// TIA Portal V16 export
// export: Created 2022-11-17T11:55:13.2880017Z, ExportSetting WithDefaults, DisplayName Totally Integrated Automation Portal, DisplayVersion V16 Update 6, DisplayName TIA Portal Version Control Interface, DisplayVersion V16 Update 2, DisplayName TIA Portal Openness, DisplayVersion V16 Update 6, DisplayName SINAMICS Startdrive Advanced, DisplayVersion V16 Update 5, DisplayName SINAMICS Startdrive G130, G150, S120, S150, SINAMICS MV, S210, DisplayVersion V16 Update 5, DisplayName SINAMICS Startdrive G110M, G120, G120C, G120D, G120P, G115D, DisplayVersion V16 Update 5, DisplayName STEP 7 Professional, DisplayVersion V16 Update 6, DisplayName STEP 7 Safety, DisplayVersion V16, DisplayName WinCC Advanced, DisplayVersion V16 Update 6
FUNCTION "FC37_MultiprogramSignal" : Void   // FC37, LAD
TITLE = Multiprogram with program selection by external signal
{ S7_Optimized_Access := 'FALSE' }
AUTHOR : Robopac
VERSION : 0.0
// stored: AutoNumber false, IsIECCheckEnabled false, SetENOAutomatically false, UDAEnableTagReadback false
   VAR_TEMP   // added for the SCL form of the ladder/FBD networks
      _w1 : Bool;
   END_VAR
BEGIN

REGION Network 1
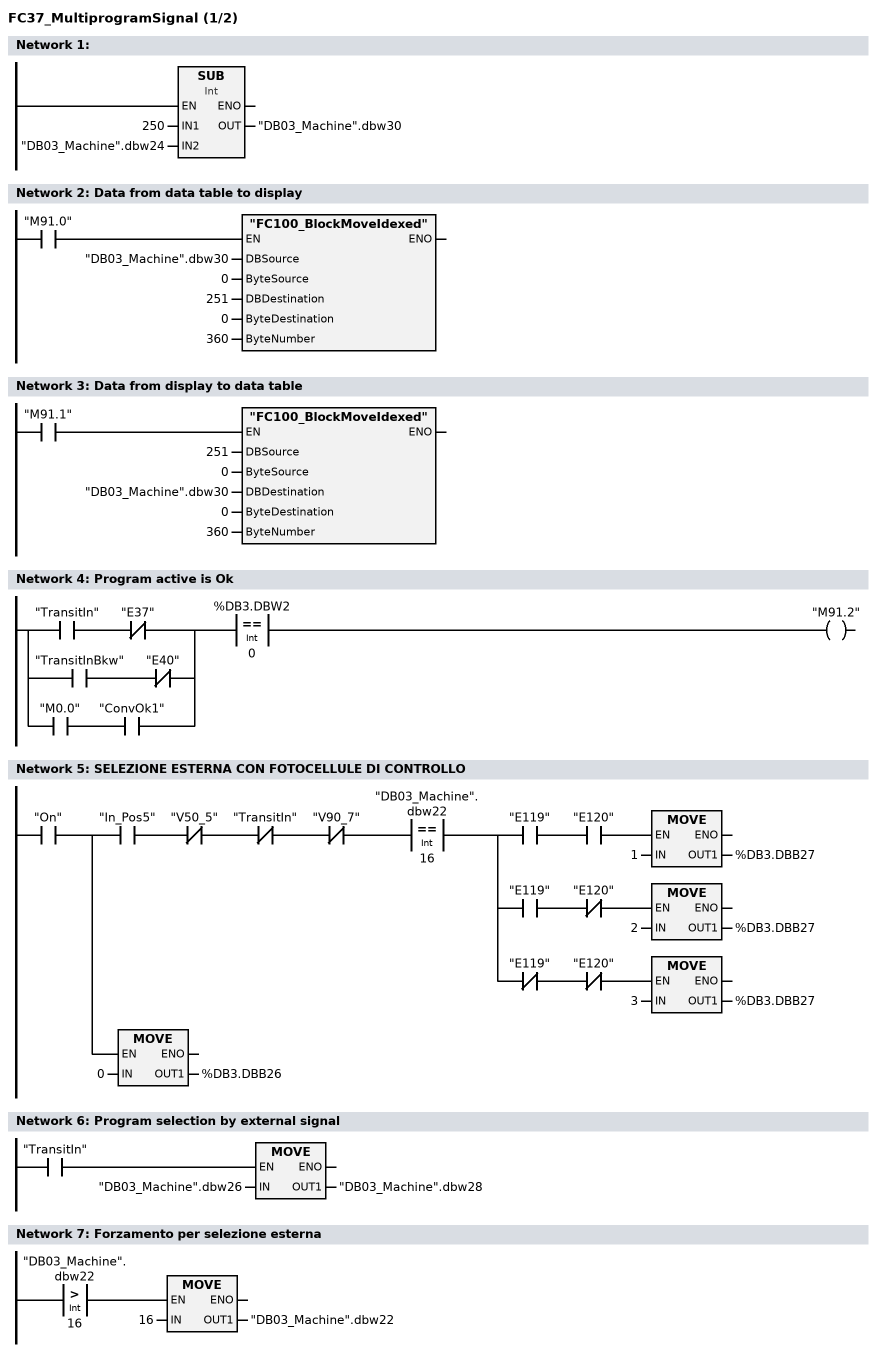
   RUNG wire#powerrail
      { S7_Templates := "SrcType := Int"; S7_GenerateENO := "TRUE" } Sub(in1 := 250, in2 := "DB03_Machine".dbw24, out => "DB03_Machine".dbw30)
   END_RUNG
   // the same network as SCL:
   "DB03_Machine".dbw30 := 250 - "DB03_Machine".dbw24;
END_REGION

REGION Network 2: Data from data table to display
   RUNG wire#powerrail
      Contact( "M91.0" )
      "FC100_BlockMoveIdexed"(DBSource := "DB03_Machine".dbw30, ByteSource := 0, DBDestination := 251, ByteDestination := 0, ByteNumber := 360)
   END_RUNG
   // the same network as SCL:
   IF "M91.0" THEN
       "FC100_BlockMoveIdexed"(DBSource := "DB03_Machine".dbw30,
                               ByteSource := 0,
                               DBDestination := 251,
                               ByteDestination := 0,
                               ByteNumber := 360);
   END_IF;
END_REGION

REGION Network 3: Data from display to data table
   RUNG wire#powerrail
      Contact( "M91.1" )
      "FC100_BlockMoveIdexed"(DBSource := 251, ByteSource := 0, DBDestination := "DB03_Machine".dbw30, ByteDestination := 0, ByteNumber := 360)
   END_RUNG
   // the same network as SCL:
   IF "M91.1" THEN
       "FC100_BlockMoveIdexed"(DBSource := 251,
                               ByteSource := 0,
                               DBDestination := "DB03_Machine".dbw30,
                               ByteDestination := 0,
                               ByteNumber := 360);
   END_IF;
END_REGION

REGION Network 4: Program active is Ok
   RUNG wire#powerrail
      Contact( "TransitIn" )
      I_Contact( "E37" )
      wire#w1
      { S7_Templates := "SrcType := Int" } EQ_Contact(in1 := %DB3.DBW2, in2 := 0)
      Coil( "M91.2" )
   END_RUNG
   RUNG wire#powerrail
      Contact( "TransitInBkw" )
      I_Contact( "E40" )
   END_RUNG wire#w1
   RUNG wire#powerrail
      Contact( "M0.0" )
      Contact( "ConvOk1" )
   END_RUNG wire#w1
   // the same network as SCL:
   "M91.2" := (("TransitIn" AND NOT "E37") OR ("TransitInBkw" AND NOT "E40") OR ("M0.0" AND "ConvOk1")) AND (%DB3.DBW2 = 0);
END_REGION

REGION Network 5: SELEZIONE ESTERNA CON FOTOCELLULE DI CONTROLLO
   RUNG wire#powerrail
      Contact( "On" )
      wire#w1
      Contact( "In_Pos5" )
      I_Contact( "V50_5" )
      I_Contact( "TransitIn" )
      I_Contact( "V90_7" )
      { S7_Templates := "SrcType := Int" } EQ_Contact(in1 := "DB03_Machine".dbw22, in2 := 16)
      wire#w2
      Contact( "E119" )
      Contact( "E120" )
      Move(in := 1, out1 => %DB3.DBB27)
   END_RUNG
   RUNG wire#w2
      Contact( "E119" )
      I_Contact( "E120" )
      Move(in := 2, out1 => %DB3.DBB27)
   END_RUNG
   RUNG wire#w2
      I_Contact( "E119" )
      I_Contact( "E120" )
      Move(in := 3, out1 => %DB3.DBB27)
   END_RUNG
   RUNG wire#w1
      { S7_GenerateENO := "TRUE" } Move(in := 0, out1 => %DB3.DBB26)
   END_RUNG
   // the same network as SCL:
   #_w1 := "On" AND "In_Pos5" AND NOT "V50_5" AND NOT "TransitIn" AND NOT "V90_7" AND ("DB03_Machine".dbw22 = 16);
   IF #_w1 AND "E119" AND "E120" THEN %DB3.DBB27 := 1; END_IF;
   IF #_w1 AND "E119" AND NOT "E120" THEN %DB3.DBB27 := 2; END_IF;
   IF #_w1 AND NOT "E119" AND NOT "E120" THEN %DB3.DBB27 := 3; END_IF;
   IF "On" THEN %DB3.DBB26 := 0; END_IF;
END_REGION

REGION Network 6: Program selection by external signal
   RUNG wire#powerrail
      Contact( "TransitIn" )
      { S7_GenerateENO := "TRUE" } Move(in := "DB03_Machine".dbw26, out1 => "DB03_Machine".dbw28)
   END_RUNG
   // the same network as SCL:
   IF "TransitIn" THEN "DB03_Machine".dbw28 := "DB03_Machine".dbw26; END_IF;
END_REGION

REGION Network 7: Forzamento per selezione esterna
   RUNG wire#powerrail
      { S7_Templates := "SrcType := Int" } GT_Contact(in1 := "DB03_Machine".dbw22, in2 := 16)
      { S7_GenerateENO := "TRUE" } Move(in := 16, out1 => "DB03_Machine".dbw22)
   END_RUNG
   // the same network as SCL:
   IF "DB03_Machine".dbw22 > 16 THEN "DB03_Machine".dbw22 := 16; END_IF;
END_REGION

REGION Network 8: Program selection by display
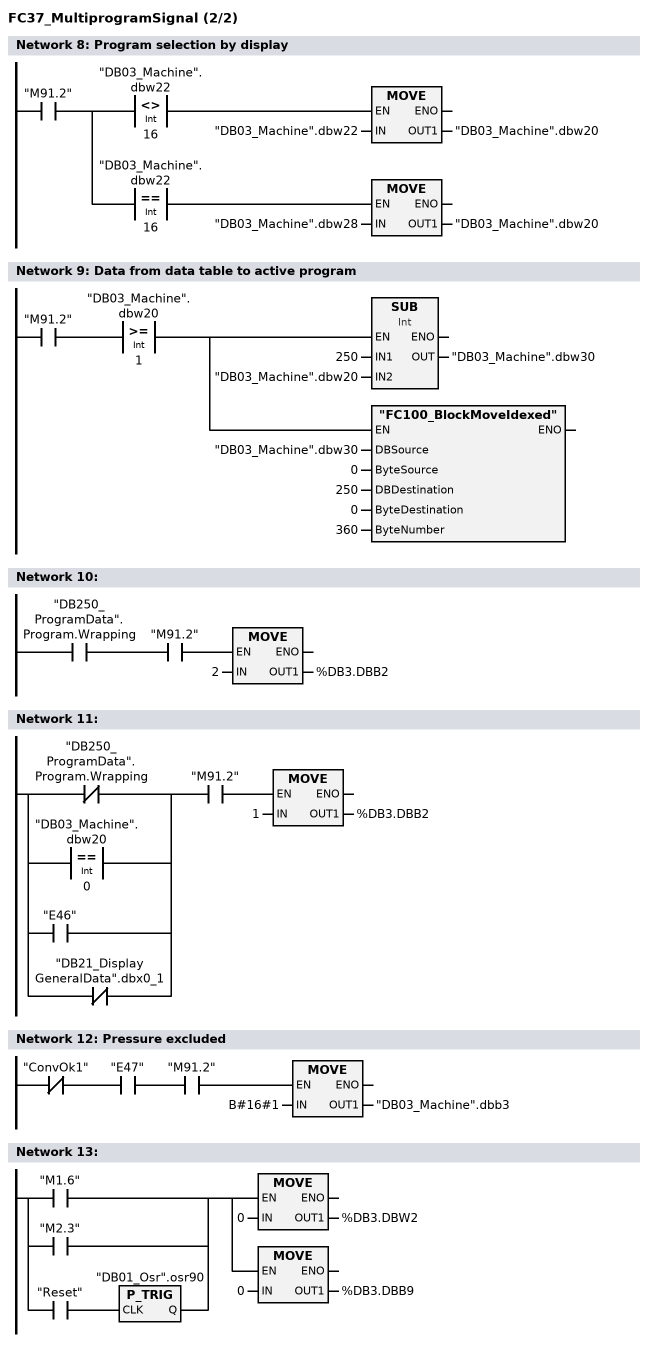
   RUNG wire#powerrail
      Contact( "M91.2" )
      wire#w1
      { S7_Templates := "SrcType := Int" } NE_Contact(in1 := "DB03_Machine".dbw22, in2 := 16)
      { S7_GenerateENO := "TRUE" } Move(in := "DB03_Machine".dbw22, out1 => "DB03_Machine".dbw20)
   END_RUNG
   RUNG wire#w1
      { S7_Templates := "SrcType := Int" } EQ_Contact(in1 := "DB03_Machine".dbw22, in2 := 16)
      { S7_GenerateENO := "TRUE" } Move(in := "DB03_Machine".dbw28, out1 => "DB03_Machine".dbw20)
   END_RUNG
   // the same network as SCL:
   IF "M91.2" AND ("DB03_Machine".dbw22 <> 16) THEN "DB03_Machine".dbw20 := "DB03_Machine".dbw22; END_IF;
   IF "M91.2" AND ("DB03_Machine".dbw22 = 16) THEN "DB03_Machine".dbw20 := "DB03_Machine".dbw28; END_IF;
END_REGION

REGION Network 9: Data from data table to active program
   RUNG wire#powerrail
      Contact( "M91.2" )
      { S7_Templates := "SrcType := Int" } GE_Contact(in1 := "DB03_Machine".dbw20, in2 := 1)
      wire#w1
      { S7_Templates := "SrcType := Int"; S7_GenerateENO := "TRUE" } Sub(in1 := 250, in2 := "DB03_Machine".dbw20, out => "DB03_Machine".dbw30)
   END_RUNG
   RUNG wire#w1
      "FC100_BlockMoveIdexed"(DBSource := "DB03_Machine".dbw30, ByteSource := 0, DBDestination := 250, ByteDestination := 0, ByteNumber := 360)
   END_RUNG
   // the same network as SCL:
   IF "M91.2" AND ("DB03_Machine".dbw20 >= 1) THEN
       "DB03_Machine".dbw30 := 250 - "DB03_Machine".dbw20;
       "FC100_BlockMoveIdexed"(DBSource := "DB03_Machine".dbw30,
                               ByteSource := 0,
                               DBDestination := 250,
                               ByteDestination := 0,
                               ByteNumber := 360);
   END_IF;
END_REGION

REGION Network 10
   RUNG wire#powerrail
      Contact( "DB250_ProgramData".Program.Wrapping )
      Contact( "M91.2" )
      { S7_GenerateENO := "TRUE" } Move(in := 2, out1 => %DB3.DBB2)
   END_RUNG
   // the same network as SCL:
   IF "DB250_ProgramData".Program.Wrapping AND "M91.2" THEN %DB3.DBB2 := 2; END_IF;
END_REGION

REGION Network 11
   RUNG wire#powerrail
      I_Contact( "DB250_ProgramData".Program.Wrapping )
      wire#w1
      Contact( "M91.2" )
      { S7_GenerateENO := "TRUE" } Move(in := 1, out1 => %DB3.DBB2)
   END_RUNG
   RUNG wire#powerrail
      { S7_Templates := "SrcType := Int" } EQ_Contact(in1 := "DB03_Machine".dbw20, in2 := 0)
   END_RUNG wire#w1
   RUNG wire#powerrail
      Contact( "E46" )
   END_RUNG wire#w1
   RUNG wire#powerrail
      I_Contact( "DB21_DisplayGeneralData".dbx0_1 )
   END_RUNG wire#w1
   // the same network as SCL:
   IF (NOT "DB250_ProgramData".Program.Wrapping OR ("DB03_Machine".dbw20 = 0) OR "E46" OR NOT "DB21_DisplayGeneralData".dbx0_1) AND "M91.2" THEN
       %DB3.DBB2 := 1;
   END_IF;
END_REGION

REGION Network 12: Pressure excluded
   RUNG wire#powerrail
      I_Contact( "ConvOk1" )
      Contact( "E47" )
      Contact( "M91.2" )
      { S7_GenerateENO := "TRUE" } Move(in := B#16#1, out1 => "DB03_Machine".dbb3)
   END_RUNG
   // the same network as SCL:
   IF NOT "ConvOk1" AND "E47" AND "M91.2" THEN "DB03_Machine".dbb3 := B#16#1; END_IF;
END_REGION

REGION Network 13
   RUNG wire#powerrail
      Contact( "M1.6" )
      wire#w1
      { S7_GenerateENO := "TRUE" } Move(in := 0, out1 => %DB3.DBW2)
   END_RUNG
   RUNG wire#powerrail
      Contact( "M2.3" )
   END_RUNG wire#w1
   RUNG wire#powerrail
      Contact( "Reset" )
      P_Trig( "DB01_Osr".osr90 )
   END_RUNG wire#w1
   RUNG wire#w1
      { S7_GenerateENO := "TRUE" } Move(in := 0, out1 => %DB3.DBB9)
   END_RUNG
   // the same network as SCL:
   #_w1 := "Reset" AND NOT "DB01_Osr".osr90;   // rising edge
   "DB01_Osr".osr90 := "Reset";
   IF "M1.6" OR "M2.3" OR #_w1 THEN
       %DB3.DBW2 := 0;
       %DB3.DBB9 := 0;
   END_IF;
END_REGION
END_FUNCTION
